FUNCTION_BLOCK DataPanel_MI_IW_CNT (* Input service interface function block for counter input data (7A/8A) *)
  (* Description: Copyright (c) 2026 HR Agrartechnik GmbH *)
  (* Version 1.0, 2026-01-17, generated, HR Agrartechnik GmbH *)
  PACKAGE DataPanel::io::MI::DI;
  IMPORT DataPanel::io::MI::const::MI;
  IMPORT DataPanel::io::MI::DI::DataPanel_MI_DI::Invalid;
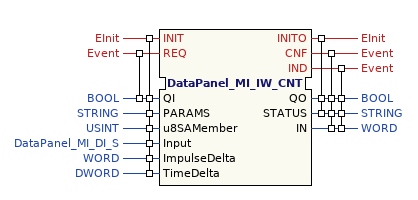
  EVENT_INPUT
    INIT : EInit WITH QI, PARAMS, u8SAMember, Input, ImpulseDelta, TimeDelta; (* Service Initialization *)
    REQ WITH QI; (* Service Request *)
  END_EVENT
  EVENT_OUTPUT
    INITO : EInit WITH QO, STATUS; (* Initialization Confirm *)
    CNF WITH QO, STATUS, IN; (* Confirmation of Requested Service *)
    IND WITH QO, STATUS, IN; (* Indication from Resource *)
  END_EVENT
  VAR_INPUT
    QI : BOOL; (* Event Input Qualifier *)
    PARAMS : STRING; (* Service Parameters *)
    u8SAMember : USINT := MI::MI_00; (* Node SA 224..239 *)
    Input : DataPanel::io::MI::DI::DataPanel_MI_DI_S := Invalid; (* Identify the Input (must be 7A or 8A) *)
    ImpulseDelta : WORD; (* After How many Impulses an IND *)
    TimeDelta : DWORD; (* After How many ms an IND *)
  END_VAR
  VAR_OUTPUT
    QO : BOOL; (* Event Output Qualifier *)
    STATUS : STRING; (* Service Status *)
    IN : WORD; (* Counter data *)
  END_VAR
END_FUNCTION_BLOCK
